Staubli VAL3: onF6Event.pgx

program onF6Event()
  local string l_sMessage
  local num l_nType
begin
  // look if the bButton is enable
  if bButton[5]
    //
    //  Clear all the List
    //
    call processList:getDefaultType(l_nType)
    logMsg("[KERNEL] INTERFACE:Clear the list")
    call processList:deleteAll(l_nType)
    if cycleStatus:bCycle
      call language:message(l_sMessage,3)
      popUpMsg(l_sMessage)
    endIf
    sEvent=""
    nIndex=0
  endIf
end
